ADAPTER IEmergencyManagement (* Adapter Interface *)
  (* Standard: 61499-1 *)
  (* Version 0.0, 11/28/2023, SESA371406, Schneider Electric *)
  PACKAGE SE.Nereda;
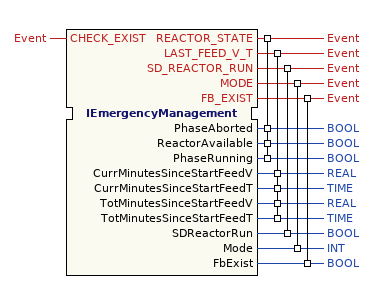
  EVENT_INPUT
    CHECK_EXIST;
  END_EVENT
  EVENT_OUTPUT
    REACTOR_STATE WITH PhaseAborted, PhaseRunning, ReactorAvailable;
    LAST_FEED_V_T WITH CurrMinutesSinceStartFeedV, CurrMinutesSinceStartFeedT, TotMinutesSinceStartFeedV, TotMinutesSinceStartFeedT;
    SD_REACTOR_RUN WITH SDReactorRun;
    MODE WITH Mode;
    FB_EXIST WITH FbExist;
  END_EVENT
  VAR_OUTPUT
    PhaseAborted : BOOL;
    ReactorAvailable : BOOL;
    PhaseRunning : BOOL;
    CurrMinutesSinceStartFeedV : REAL;
    CurrMinutesSinceStartFeedT : TIME;
    TotMinutesSinceStartFeedV : REAL;
    TotMinutesSinceStartFeedT : TIME;
    SDReactorRun : BOOL;
    Mode : INT;
    FbExist : BOOL;
  END_VAR
  SERVICE SOCKET/PLUG
    SEQUENCE request_confirm
      SOCKET.REQ(REQD) -> PLUG.REQ(REQD);
      PLUG.CNF(CNFD) -> SOCKET.CNF(CNFD);
    END_SEQUENCE
    SEQUENCE indication_response
      PLUG.IND(INDD) -> SOCKET.IND(INDD);
      SOCKET.RSP(RSPD) -> PLUG.RSP(RSPD);
    END_SEQUENCE
  END_SERVICE
END_ADAPTER
